// TIA Portal V20 export
DATA_BLOCK "DataToSafety"   // DB120
// stored: Access Published, InstanceOfName Safety.typeDataToSafety, InstanceOfType UDT, Namespace Safety
"Safety.typeDataToSafety"
   // VAR
   //    ackSafetyFromHmi : Int;
   //    ackSafetyGlobal : Bool;
   //    ackFromUnit1 : Bool;
   //    ackSafetyFromMobileHMI : Bool;
   //    resetSafetyFromMobileHMI : Bool;
   //    connectionBoxID_1 : Int;
   //    connectionBoxID_2 : Int;
   //    MobilePanelConnected : Bool;
   //    MobilePanelPermissions : Bool;
   //    DeselectBA10 : Bool;
   //    DeselectBA15 : Bool;
   //    DeselectBA30 : Bool;
   //    DeselectBA60 : Bool;
   //    PowerOnCommand : Bool;
   //    InitializeEnable : Bool;   // Main OP Home
   //    BA060STOP : Bool;
   //    SepaGripperAxisXmoveToBa60 : Bool;
   //    unitMode : "Safety.typeUnitMode";
   //    unitState : "Safety.typeUnitStatus";
   //    winderUsed : "Safety.typeWinderUseMode";
   //    StackDoor1 { S7_SetPoint := 'True'} : "Safety.typeFdoorCommands";
   //    StackDoor2 { S7_SetPoint := 'True'} : "Safety.typeFdoorCommands";
   //    StackDoor3 { S7_SetPoint := 'True'} : "Safety.typeFdoorCommands";
   //    StackDoor4 { S7_SetPoint := 'True'} : "Safety.typeFdoorCommands";
   //    StackDoor5 { S7_SetPoint := 'True'} : "Safety.typeFdoorCommands";
   //    StackDoor6 { S7_SetPoint := 'True'} : "Safety.typeFdoorCommands";
   //    StackDoor7 { S7_SetPoint := 'True'} : "Safety.typeFdoorCommands";
   //    StackDoor8 { S7_SetPoint := 'True'} : "Safety.typeFdoorCommands";
   //    StackDoor9 { S7_SetPoint := 'True'} : "Safety.typeFdoorCommands";
   //    StackDoor10 { S7_SetPoint := 'True'} : "Safety.typeFdoorCommands";
   //    StackDoor12 { S7_SetPoint := 'True'} : "Safety.typeFdoorCommands";
   //    hotWireCutterCmds : "Safety.typeHotWireCutter";
   //    clock { ExternalAccessible := 'False'; ExternalVisible := 'False'; ExternalWritable := 'False'} : "Safety.typeGlobalClockMem";
   //    BrakeTest { S7_SetPoint := 'True'} : "Safety.typeBrakeTest";
   // END_VAR
BEGIN
END_DATA_BLOCK
